% RSLogix 500 project FINAL.RSS, saved by version 8.30.00.16 %
PROJECT "UNTITLED"    % processor: Bul.1763 MicroLogix 1100 Series B %

PROGRAM FILES
  LAD 2 "MAIN"  3 rungs
  LAD 3 "DIGITAL IO"  8 rungs
  LAD 4 "CTRL LOGIC"  23 rungs

DATA FILES
  O0 OUTPUT  5 elements
  I1 INPUT  7 elements
  S2 STATUS  66 elements
  B3 BINARY  8 elements
  T4 TIMER  9 elements
  C5 COUNTER  1 elements
  R6 CONTROL  1 elements
  N7 INTEGER  1 elements
  F8 FLOAT  1 elements

LADDER 2 "MAIN"
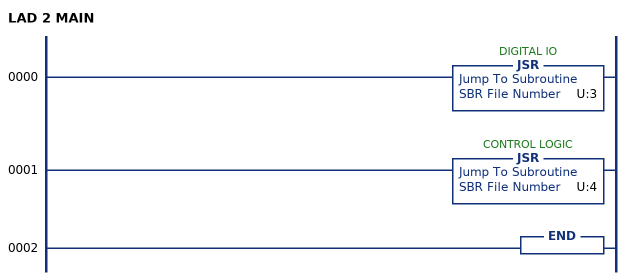
% Rung: 0 %
SOR JSR U:3 EOR
%   U:3  "DIGITAL IO" %
% Rung: 1 %
SOR JSR U:4 EOR
%   U:4  "CONTROL LOGIC" %
% Rung: 2 %
SOR END EOR

LADDER 3 "DIGITAL IO"
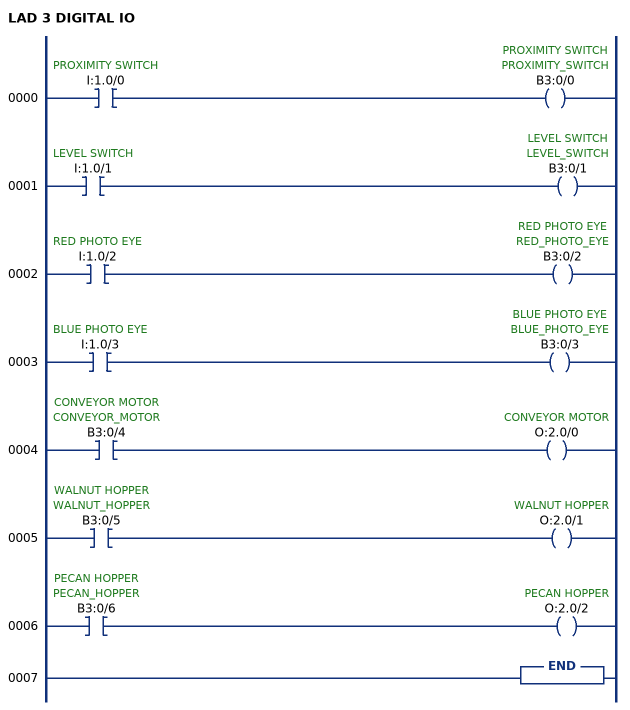
% Rung: 0 %
SOR XIC I:1.0/0 OTE B3:0/0 EOR
%   I:1.0/0  "PROXIMITY SWITCH" %
%   B3:0/0  PROXIMITY_SWITCH  "PROXIMITY SWITCH" %
% Rung: 1 %
SOR XIC I:1.0/1 OTE B3:0/1 EOR
%   I:1.0/1  "LEVEL SWITCH" %
%   B3:0/1  LEVEL_SWITCH  "LEVEL SWITCH" %
% Rung: 2 %
SOR XIC I:1.0/2 OTE B3:0/2 EOR
%   I:1.0/2  "RED PHOTO EYE" %
%   B3:0/2  RED_PHOTO_EYE  "RED PHOTO EYE" %
% Rung: 3 %
SOR XIC I:1.0/3 OTE B3:0/3 EOR
%   I:1.0/3  "BLUE PHOTO EYE" %
%   B3:0/3  BLUE_PHOTO_EYE  "BLUE PHOTO EYE" %
% Rung: 4 %
SOR XIC B3:0/4 OTE O:2.0/0 EOR
%   B3:0/4  CONVEYOR_MOTOR  "CONVEYOR MOTOR" %
%   O:2.0/0  "CONVEYOR MOTOR" %
% Rung: 5 %
SOR XIC B3:0/5 OTE O:2.0/1 EOR
%   B3:0/5  WALNUT_HOPPER  "WALNUT HOPPER" %
%   O:2.0/1  "WALNUT HOPPER" %
% Rung: 6 %
SOR XIC B3:0/6 OTE O:2.0/2 EOR
%   B3:0/6  PECAN_HOPPER  "PECAN HOPPER" %
%   O:2.0/2  "PECAN HOPPER" %
% Rung: 7 %
SOR END EOR

LADDER 4 "CTRL LOGIC"
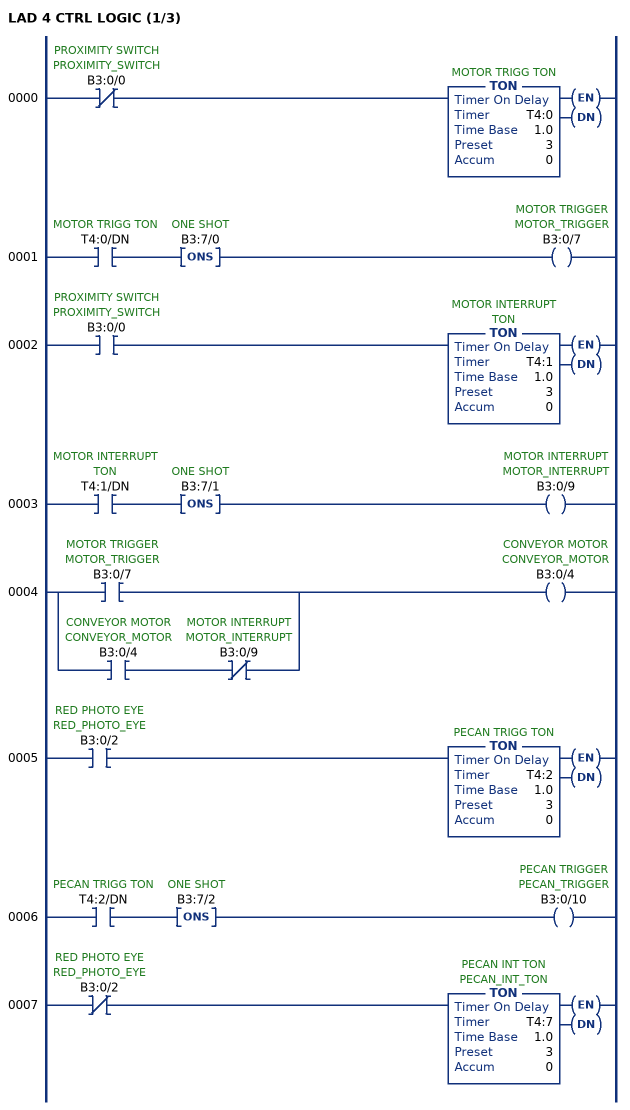
% Rung: 0 %
SOR XIO B3:0/0 TON T4:0 1.0 3 0 EOR
%   B3:0/0  PROXIMITY_SWITCH  "PROXIMITY SWITCH" %
%   T4:0  "MOTOR TRIGG TON" %
% Rung: 1 %
SOR XIC T4:0/DN ONS B3:7/0 OTE B3:0/7 EOR
%   T4:0  "MOTOR TRIGG TON" %
%   B3:7/0  "ONE SHOT" %
%   B3:0/7  MOTOR_TRIGGER  "MOTOR TRIGGER" %
% Rung: 2 %
SOR XIC B3:0/0 TON T4:1 1.0 3 0 EOR
%   B3:0/0  PROXIMITY_SWITCH  "PROXIMITY SWITCH" %
%   T4:1  "MOTOR INTERRUPT TON" %
% Rung: 3 %
SOR XIC T4:1/DN ONS B3:7/1 OTE B3:0/9 EOR
%   T4:1/DN  "MOTOR INTERRUPT TON" %
%   B3:7/1  "ONE SHOT" %
%   B3:0/9  MOTOR_INTERRUPT  "MOTOR INTERRUPT" %
% Rung: 4 %
SOR BST XIC B3:0/7 NXB XIC B3:0/4 XIO B3:0/9 BND OTE B3:0/4 EOR
%   B3:0/7  MOTOR_TRIGGER  "MOTOR TRIGGER" %
%   B3:0/4  CONVEYOR_MOTOR  "CONVEYOR MOTOR" %
%   B3:0/9  MOTOR_INTERRUPT  "MOTOR INTERRUPT" %
% Rung: 5 %
SOR XIC B3:0/2 TON T4:2 1.0 3 0 EOR
%   B3:0/2  RED_PHOTO_EYE  "RED PHOTO EYE" %
%   T4:2  "PECAN TRIGG TON" %
% Rung: 6 %
SOR XIC T4:2/DN ONS B3:7/2 OTE B3:0/10 EOR
%   T4:2  "PECAN TRIGG TON" %
%   B3:7/2  "ONE SHOT" %
%   B3:0/10  PECAN_TRIGGER  "PECAN TRIGGER" %
% Rung: 7 %
SOR XIO B3:0/2 TON T4:7 1.0 3 0 EOR
%   B3:0/2  RED_PHOTO_EYE  "RED PHOTO EYE" %
%   T4:7  PECAN_INT_TON  "PECAN INT TON" %

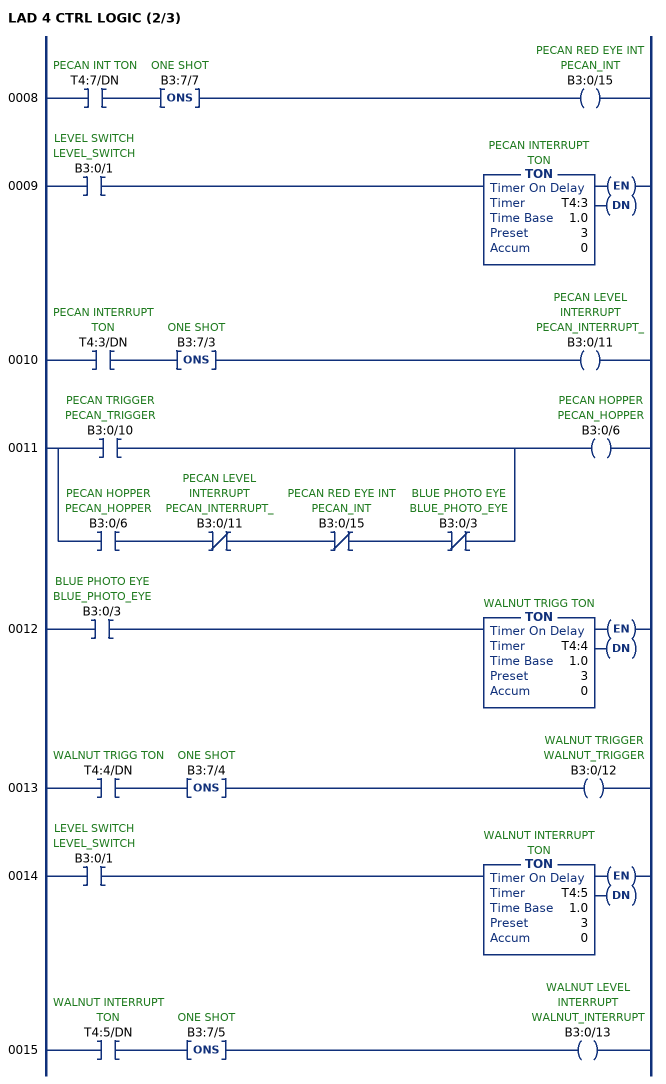
% Rung: 8 %
SOR XIC T4:7/DN ONS B3:7/7 OTE B3:0/15 EOR
%   T4:7/DN  "PECAN INT TON" %
%   B3:7/7  "ONE SHOT" %
%   B3:0/15  PECAN_INT  "PECAN RED EYE INT" %
% Rung: 9 %
SOR XIC B3:0/1 TON T4:3 1.0 3 0 EOR
%   B3:0/1  LEVEL_SWITCH  "LEVEL SWITCH" %
%   T4:3  "PECAN INTERRUPT TON" %
% Rung: 10 %
SOR XIC T4:3/DN ONS B3:7/3 OTE B3:0/11 EOR
%   T4:3  "PECAN INTERRUPT TON" %
%   B3:7/3  "ONE SHOT" %
%   B3:0/11  PECAN_INTERRUPT_  "PECAN LEVEL INTERRUPT" %
% Rung: 11 %
SOR BST XIC B3:0/10 NXB XIC B3:0/6 XIO B3:0/11 XIO B3:0/15 XIO B3:0/3 BND OTE B3:0/6 EOR
%   B3:0/10  PECAN_TRIGGER  "PECAN TRIGGER" %
%   B3:0/6  PECAN_HOPPER  "PECAN HOPPER" %
%   B3:0/11  PECAN_INTERRUPT_  "PECAN LEVEL INTERRUPT" %
%   B3:0/15  PECAN_INT  "PECAN RED EYE INT" %
%   B3:0/3  BLUE_PHOTO_EYE  "BLUE PHOTO EYE" %
% Rung: 12 %
SOR XIC B3:0/3 TON T4:4 1.0 3 0 EOR
%   B3:0/3  BLUE_PHOTO_EYE  "BLUE PHOTO EYE" %
%   T4:4  "WALNUT TRIGG TON" %
% Rung: 13 %
SOR XIC T4:4/DN ONS B3:7/4 OTE B3:0/12 EOR
%   T4:4  "WALNUT TRIGG TON" %
%   B3:7/4  "ONE SHOT" %
%   B3:0/12  WALNUT_TRIGGER  "WALNUT TRIGGER" %
% Rung: 14 %
SOR XIC B3:0/1 TON T4:5 1.0 3 0 EOR
%   B3:0/1  LEVEL_SWITCH  "LEVEL SWITCH" %
%   T4:5  "WALNUT INTERRUPT TON" %
% Rung: 15 %
SOR XIC T4:5/DN ONS B3:7/5 OTE B3:0/13 EOR
%   T4:5  "WALNUT INTERRUPT TON" %
%   B3:7/5  "ONE SHOT" %
%   B3:0/13  WALNUT_INTERRUPT  "WALNUT LEVEL INTERRUPT" %

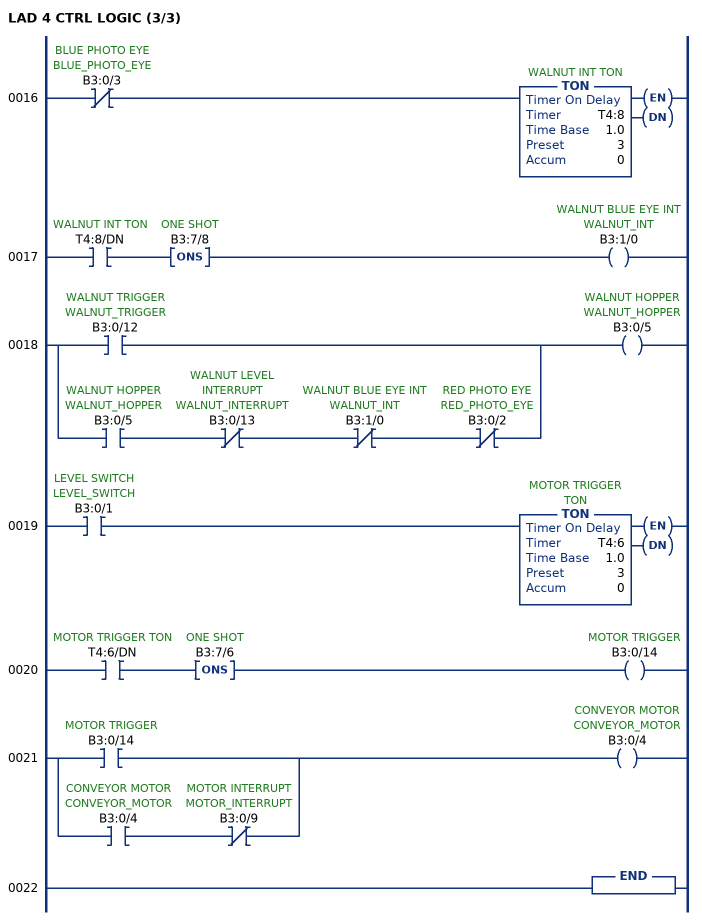
% Rung: 16 %
SOR XIO B3:0/3 TON T4:8 1.0 3 0 EOR
%   B3:0/3  BLUE_PHOTO_EYE  "BLUE PHOTO EYE" %
%   T4:8  "WALNUT INT TON" %
% Rung: 17 %
SOR XIC T4:8/DN ONS B3:7/8 OTE B3:1/0 EOR
%   T4:8  "WALNUT INT TON" %
%   B3:7/8  "ONE SHOT" %
%   B3:1/0  WALNUT_INT  "WALNUT BLUE EYE INT" %
% Rung: 18 %
SOR BST XIC B3:0/12 NXB XIC B3:0/5 XIO B3:0/13 XIO B3:1/0 XIO B3:0/2 BND OTE B3:0/5 EOR
%   B3:0/12  WALNUT_TRIGGER  "WALNUT TRIGGER" %
%   B3:0/5  WALNUT_HOPPER  "WALNUT HOPPER" %
%   B3:0/13  WALNUT_INTERRUPT  "WALNUT LEVEL INTERRUPT" %
%   B3:1/0  WALNUT_INT  "WALNUT BLUE EYE INT" %
%   B3:0/2  RED_PHOTO_EYE  "RED PHOTO EYE" %
% Rung: 19 %
SOR XIC B3:0/1 TON T4:6 1.0 3 0 EOR
%   B3:0/1  LEVEL_SWITCH  "LEVEL SWITCH" %
%   T4:6  "MOTOR TRIGGER TON" %
% Rung: 20 %
SOR XIC T4:6/DN ONS B3:7/6 OTE B3:0/14 EOR
%   T4:6  "MOTOR TRIGGER TON" %
%   B3:7/6  "ONE SHOT" %
%   B3:0/14  "MOTOR TRIGGER" %
% Rung: 21 %
SOR BST XIC B3:0/14 NXB XIC B3:0/4 XIO B3:0/9 BND OTE B3:0/4 EOR
%   B3:0/14  "MOTOR TRIGGER" %
%   B3:0/4  CONVEYOR_MOTOR  "CONVEYOR MOTOR" %
%   B3:0/9  MOTOR_INTERRUPT  "MOTOR INTERRUPT" %
% Rung: 22 %
SOR END EOR

OTHER DOCUMENTED ADDRESSES
  B3:0/8  "ONE SHOT"
  I:1.0  "PROXIMITY SWITCH"
  I:1.1  "LEVEL SWITCH"
  I:1.2  "RED PHOTO EYE"
  I:1.3  "BLUE PHOTO EYE"
  O:2.0  "CONVEYOR MOTOR"
  O:2.1  "WALNUT HOPPER"
  O:2.2  "PECAN HOPPER"

DATA TABLE (non-zero values as saved)
DATA T4
% .PRE .ACC %
% T4:0 % 3 0
% T4:1 % 3 0
% T4:2 % 3 0
% T4:3 % 3 0
% T4:4 % 3 0
% T4:5 % 3 0
% T4:6 % 3 0
% T4:7 % 3 0
% T4:8 % 3 0
